INTERFACE I_Command

METHOD Execute
END_METHOD

END_INTERFACE

(* stored: Version 1.1.0.1, ProductVersion 3.1.4024.12
   Itf I_Command: Id {a1d5eca1-cdce-4e7c-a011-6f83ce7d8fde}
   Method Execute: Id {cf6b983e-7795-47db-8569-b6a04918d1f3} *)
